FUNCTION_BLOCK ModelLightSet (* Composite Function Block Type *)
  (* Standard: 61499-2 *)
  (* Version 0.2, 2003-12-05, JHC, Rockwell Automation, Renamed from NEWCOMPFB. *)
  (* Version 0.1, 2002-01-08, JHC, Rockwell Automation, Added DLY FB as example. *)
  (* Version 0.0, 2000-05-27, JHC, Rockwell Automation *)
  (* Compiler header: package fb.rt.Assingment; *)
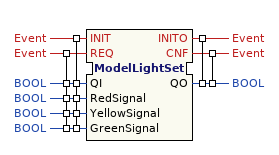
  EVENT_INPUT
    INIT WITH QI, RedSignal, YellowSignal, GreenSignal; (* Initialization Request *)
    REQ WITH QI, RedSignal, YellowSignal, GreenSignal; (* Normal Execution Request *)
  END_EVENT
  EVENT_OUTPUT
    INITO WITH QO; (* Initialization Confirm *)
    CNF WITH QO; (* Execution Confirmation *)
  END_EVENT
  VAR_INPUT
    QI : BOOL; (* Input event qualifier *)
    RedSignal : BOOL;
    YellowSignal : BOOL;
    GreenSignal : BOOL;
  END_VAR
  VAR_OUTPUT
    QO : BOOL; (* Output event qualifier *)
  END_VAR
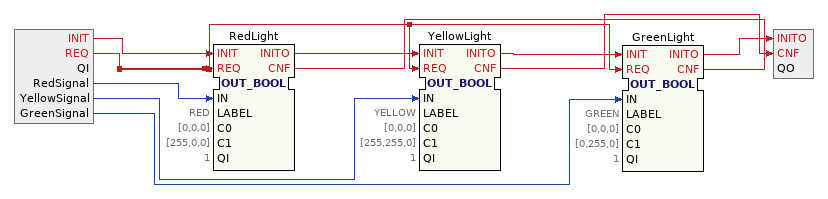
  FBS
    RedLight : OUT_BOOL(LABEL := RED, C0 := [0,0,0], C1 := [255,0,0], QI := 1);
    YellowLight : OUT_BOOL(LABEL := YELLOW, C0 := [0,0,0], C1 := [255,255,0], QI := 1);
    GreenLight : OUT_BOOL(LABEL := GREEN, C0 := [0,0,0], C1 := [0,255,0], QI := 1);
  END_FBS
  EVENT_CONNECTIONS
    RedLight.INITO TO YellowLight.INIT;
    YellowLight.INITO TO GreenLight.INIT;
    INIT TO RedLight.INIT;
    GreenLight.INITO TO INITO;
    REQ TO RedLight.REQ;
    REQ TO YellowLight.REQ;
    REQ TO GreenLight.REQ;
    RedLight.CNF TO CNF;
    YellowLight.CNF TO CNF;
    GreenLight.CNF TO CNF;
  END_CONNECTIONS
  DATA_CONNECTIONS
    RedSignal TO RedLight.IN;
    YellowSignal TO YellowLight.IN;
    GreenSignal TO GreenLight.IN;
  END_CONNECTIONS
END_FUNCTION_BLOCK
